FUNCTION_BLOCK FB_Regelingen
VAR_INPUT
    BestuurMode : INT;            (* 0 = Handmatig, 1 = Automatisch *)
    RegelStand1 : REAL;           (* Setpoint debiet in m³/s *)
    RegelStand2 : REAL;           (* Setpoint polderpeil in m NAP *)
    Mode : INT;                   (* 0 = Uit, 1 = Polderpeil, 2 = Constant Debiet *)
    CurrentPosition : REAL;       (* Terugmelding analoog *)
    DeltaH : REAL;                (* Niveauverschil *)
END_VAR

// Output naar andere functieblokken
VAR_OUTPUT
    OpenSignal : BOOL;
    CloseSignal : BOOL;
    FlowRate : REAL;
END_VAR

VAR
    (* Uitgangen *)
    Pomp1 : INT;                  (* Status pomp 1: 0 = uit, 1 = aan *)
    Pomp2 : INT;                  (* Status pomp 2: 0 = uit, 1 = aan *)

    (* Interne variabelen *)
    ModeStatus : STRING[20];      (* Beschrijft huidige modus *)
    ActiveStand : STRING[20];     (* Beschrijft actieve regelstand *)

    (* Instanties van subfunctieblokken *)
    Uitlaten : FB_Uitlaten;
    Uitmalen : FB_Uitmalen;
    Inmalen : FB_Inmalen;

    (* Interne statusbewaking *)
    DebietError : REAL;           (* Foutwaarde van debietregeling *)
    PolderpeilError : REAL;       (* Foutwaarde van polderpeilregeling *)

    (* Variabelen voor pompberekeningen *)
    berekendeRPM_REAL : LREAL;
    berekendeRPM_UINT : UINT;
    M2021_ON : BOOL;
    stuurRPM_M2021 : UINT;
    currentRPM_M2021 : UINT;
    minRPM_M2021 : UINT := 20;
    maxRPM_M2021 : UINT := 1000;
    P2021_status : BOOL;
    P2021_setpoint : UINT;
    P2021_stand : INT;            (* 1 = actief, 0 = uit *)
    polderHoogteVerschil : REAL;  (* Hoogteverschil in meters *)

    (* Variabelen voor pomp 2 berekening *)
    berekendeRPM2_REAL : LREAL;
    berekendeRPM2_UINT : UINT;
    M2011_ON : BOOL;
    stuurRPM_M2011 : UINT;
    currentRPM_M2011 : UINT;
    minRPM_M2011 : UINT := 20;
    maxRPM_M2011 : UINT := 1000;
    P2011_status : BOOL;
    P2011_setpoint : UINT;
    P2011_stand : INT;            (* 1 = actief, 0 = uit *)
    zomerPijl : BOOL;
    streefPijl : REAL;

    (* Methodes voor regeling *)
    TargetPosition : REAL;
    Timer : TON;
    CD : REAL := 0.82;
    G : REAL := 9.81;
    Area : REAL;
    currentStateRegeling: E_RegelingState;
    MaxPosition: REAL;
    MinPosition: REAL;
    MinSpeed: REAL;
    NominalSpeed: REAL;
    MaxSpeed: REAL;
    H0: REAL;
	Q0: REAL;
	MaxSchuifArea: REAL;
	CalculatePositionForFlow: REAL;
	CalculateSpeedForFlow: REAL;
END_VAR

CASE BestuurMode OF
    0:  // Handmatige modus
        // Zet alle uitvoer naar een veilige stand
        OpenSignal := FALSE;
        CloseSignal := FALSE;
        FlowRate := 0.0;

    1:  // Automatische modus
        CASE currentStateRegeling OF
            E_RegelingState.uit:
                // Roep de `Uit`-methode aan
                Uit();
                // Zet alle uitvoer naar veilige stand in de 'uit' modus
                FlowRate := 0.0;
                OpenSignal := FALSE;
                CloseSignal := TRUE;

            E_RegelingState.polderpeil:
                // Roep de `Polderpeil`-methode aan voor het regelen van het waterpeil
                FlowRate := Polderpeil(DeltaH, MaxPosition, MinPosition, currentStateRegeling, MinSpeed, NominalSpeed, MaxSpeed, H0);
                // Controleer of de klep open of gesloten moet zijn op basis van de flowrate
                OpenSignal := (FlowRate > 0.0);
                CloseSignal := NOT OpenSignal;

            E_RegelingState.debiet:
    // Roep de `Debiet`-methode aan voor het regelen van het debiet
    FlowRate := Debiet(RegelStand1, DeltaH, Q0, H0, NominalSpeed, MaxSpeed, MinSpeed, CD, G, Area, MaxSchuifArea, CalculatePositionForFlow, CalculateSpeedForFlow);
    // Controleer of de klep open of gesloten moet zijn op basis van de flowrate
    OpenSignal := (FlowRate > 0.0);
    CloseSignal := NOT OpenSignal;
	
        END_CASE;
END_CASE;

// Zorg ervoor dat de signaalwaarden (OpenSignal, CloseSignal) doorgegeven worden naar de andere functieblokken
Uitlaten.FlowRate := FlowRate; // Doorgeven van de FlowRate naar FB_Uitlaten
Uitlaten.OpenSignal := OpenSignal; // Doorgeven van OpenSignal naar FB_Uitlaten
Uitlaten.CloseSignal := CloseSignal; // Doorgeven van CloseSignal naar FB_Uitlaten

Uitmalen.FlowRate := FlowRate; // Doorgeven van de FlowRate naar FB_Uitmalen
Uitmalen.OpenSignal := OpenSignal; // Doorgeven van OpenSignal naar FB_Uitmalen
Uitmalen.CloseSignal := CloseSignal; // Doorgeven van CloseSignal naar FB_Uitmalen

// Voeg eventueel de logica voor andere functieblokken toe, zoals FB_Inmalen

METHOD Debiet : REAL
VAR_INPUT
    DesiredFlow : REAL;           (* Het gewenste debiet in m³/s *)
    DeltaH : REAL;                (* Niveauverschil *)
    Q0 : REAL := 1.26;            (* Referentiedebiet *)
    H0 : REAL := 3.42;            (* Referentiehoogte *)
    NominalSpeed : REAL := 321.0; (* Nominale snelheid van de pomp *)
    MaxSpeed : REAL := 350.0;     (* Maximale snelheid van de pomp *)
    MinSpeed : REAL := 100.0;     (* Minimale snelheid van de pomp *)
    CD : REAL := 0.82;            (* Coëfficiënt van de pomp *)
    G : REAL := 9.81;             (* Gravitatieversnelling *)
    Area : REAL;                  (* Oppervlakte van de schuif *)
    MaxSchuifArea : REAL := 1.0;  (* Maximale schuifopendiameter *)
    CalculatePositionForFlow : REAL; (* Berekening van de positie op basis van debiet *)
    CalculateSpeedForFlow : REAL;   (* Berekening van de snelheid op basis van debiet *)
END_VAR

VAR
    FlowRate : REAL;             (* Het berekende debiet *)
    SpeedForFlow : REAL;         (* De snelheid op basis van het debiet *)
    PositionForFlow : REAL;      (* De positie op basis van het debiet *)
END_VAR
(* Bereken de FlowRate op basis van het niveauverschil en andere parameters *)
IF DeltaH > 0 THEN
    Area := DesiredFlow / (CD * SQRT(2 * G * DeltaH));  (* Bereken de benodigde oppervlakte *)
    PositionForFlow := Area / MaxSchuifArea;              (* Bereken de positie voor het debiet *)
    SpeedForFlow := NominalSpeed * SQRT(DesiredFlow / Q0 + DeltaH / H0); (* Bereken de snelheid *)

    (* Beperk de snelheid binnen de limieten van de pomp *)
    IF SpeedForFlow > MaxSpeed THEN
        SpeedForFlow := MaxSpeed; 
    ELSIF SpeedForFlow < MinSpeed THEN
        SpeedForFlow := MinSpeed; 
    END_IF;

    (* Het debiet wordt berekend *)
    FlowRate := SpeedForFlow * Area; (* Bereken het debiet met de opgegeven snelheid en oppervlakte *)

ELSE
    (* Als het niveauverschil nul of negatief is, wordt het debiet als nul beschouwd *)
    PositionForFlow := 0.0;
    SpeedForFlow := MinSpeed;  (* Stel de snelheid in op de minimale snelheid *)
    FlowRate := 0.0;          (* Het debiet is nul bij negatieve of nul DeltaH *)
END_IF;

(* Teruggeven van de berekende debiet *)
Debiet := FlowRate;
END_METHOD

METHOD Polderpeil : REAL
VAR_INPUT
    DeltaH : REAL; 
    MaxPosition : REAL := 1.0;  // Maximale positie
    MinPosition : REAL := 0.0;  // Minimale positie
    currentStateRegeling: E_RegelingState;
    MinSpeed : REAL := 100.0;  // Minimale snelheid
    NominalSpeed : REAL := 321.0;  // Nominale snelheid
    MaxSpeed : REAL := 350.0;  // Maximale snelheid
    H0 : REAL := 3.42;  // Referentiehoogte
END_VAR

VAR
    CalculatePositionForWaterLevel : REAL;  // Berekende positie voor waterpeil
    CalculateSpeedForWaterLevel : REAL;     // Berekende snelheid voor waterpeil
END_VAR
// Berekeningen voor het waterpeil
IF DeltaH > 0 THEN
    // Bereken de snelheid en positie voor het waterpeil
    CalculateSpeedForWaterLevel := MinSpeed + (NominalSpeed - MinSpeed) * (DeltaH / H0);
    CalculatePositionForWaterLevel := MinPosition + (MaxPosition - MinPosition) * (DeltaH / 1.0); 
    
    // Beperk de snelheid tot de maximale waarde
    IF CalculateSpeedForWaterLevel > MaxSpeed THEN
        CalculateSpeedForWaterLevel := MaxSpeed; 
    END_IF;
ELSE
    // Zet de positie en snelheid naar de minimale waarden als het niveauverschil niet positief is
    CalculatePositionForWaterLevel := MinPosition; 
    CalculateSpeedForWaterLevel := MinSpeed;
END_IF;

// Retourneer de berekende snelheid voor gebruik in de regeling
RETURN CalculateSpeedForWaterLevel;
END_METHOD

PROPERTY Statusdebiet : E_RegelingState
GET
END_GET
SET
END_SET
END_PROPERTY

PROPERTY StatusPolderpeil : E_RegelingState
GET
END_GET
SET
END_SET
END_PROPERTY

PROPERTY Statusuit : E_RegelingState
SET
END_SET
END_PROPERTY

METHOD Uit : VOID
VAR
    currentStateregeling: E_REGELINGSTATE;
    PumpOn: BOOL;
    DesiredSpeed: REAL;
    OpenSignal: BOOL;
    CloseSignal: BOOL;
END_VAR
// Controleer of de regeling in de "Uit" stand staat
IF currentStateregeling = E_RegelingState.uit THEN
    // Zet de pompen uit
    PumpOn := FALSE;  // Pompstatus uitzetten

    // Zet de gewenste snelheid naar 0 (geen beweging)
    DesiredSpeed := 0.0;

    // Zet de kleppen uit
    OpenSignal := FALSE;  // Geen open signaal voor de kleppen
    CloseSignal := TRUE;  // Sluit de kleppen
    
    // Extra actie kan hier toegevoegd worden (bijvoorbeeld reset van andere systemen)
END_IF
END_METHOD

END_FUNCTION_BLOCK

(* stored: Version 1.1.0.1, ProductVersion 3.1.4026.8
   POU FB_Regelingen: Id {10454be2-17f1-45a6-927c-6671ec7f7806}, SpecialFunc None
   Folder Methods: Id {7a5154a8-d0ab-4aca-a913-d3242cae32ca}
   Folder Properties: Id {64d43a35-4d5a-4d04-a035-1c51de5047d0}
   Method Debiet: Id {2b69d816-b4da-4e63-b57a-877adece09f6}
   Method Polderpeil: Id {4de05532-21a1-4e5c-8e2d-3a2285633ff7}
   Property Statusdebiet: Id {27f04e5c-872c-417b-b202-7a7edac38bfd}
   Get Get: Id {0df83d80-bdac-4b44-bc88-00d562838eb3}
   Set Set: Id {c175d2e1-d2b4-4540-a5e4-9545957390d2}
   Property StatusPolderpeil: Id {32e1e152-1b90-473e-b502-821a058bfe88}
   Get Get: Id {7201f6cb-5b60-4ee4-b9b6-21f564618a85}
   Set Set: Id {b9b5e7b8-ea12-4383-8890-4ea40e547a06}
   Property Statusuit: Id {ccfa43fa-e8bd-4c2a-804c-d61e6c9e0d26}
   Set Set: Id {0512026f-e1fd-4f9b-9f3b-27d1457d7276}
   Method Uit: Id {09b90ffb-84c9-47ca-b34d-35c9241a6e0a} *)
